TYPE E_MesgSevr :
(
	Info := 0,
	Debug	:= 1,
	Warning	:= 2,
	Fault	:= 3
	
);
END_TYPE

(* stored: Version 1.1.0.1, ProductVersion 3.1.4018.5
   DUT E_MesgSevr: Id {cb5c14c3-fbb9-40ae-b518-0fced558f634} *)
